% RSLogix 500 project JOB 13 UN FIN_BAK035.RSS, saved by version 10.00.00.00 %
PROJECT "ML06B"    % processor: Bul.1763 MicroLogix 1100 Series B %

PROGRAM FILES
  LAD 2   13 rungs

DATA FILES
  O0 OUTPUT  4 elements
  I1 INPUT  6 elements
  S2 STATUS  66 elements
  B3 BINARY  1 elements
  T4 TIMER  1 elements
  C5 COUNTER  1 elements
  R6 CONTROL  1 elements
  N7 INTEGER  1 elements
  F8 FLOAT  1 elements

LADDER 2
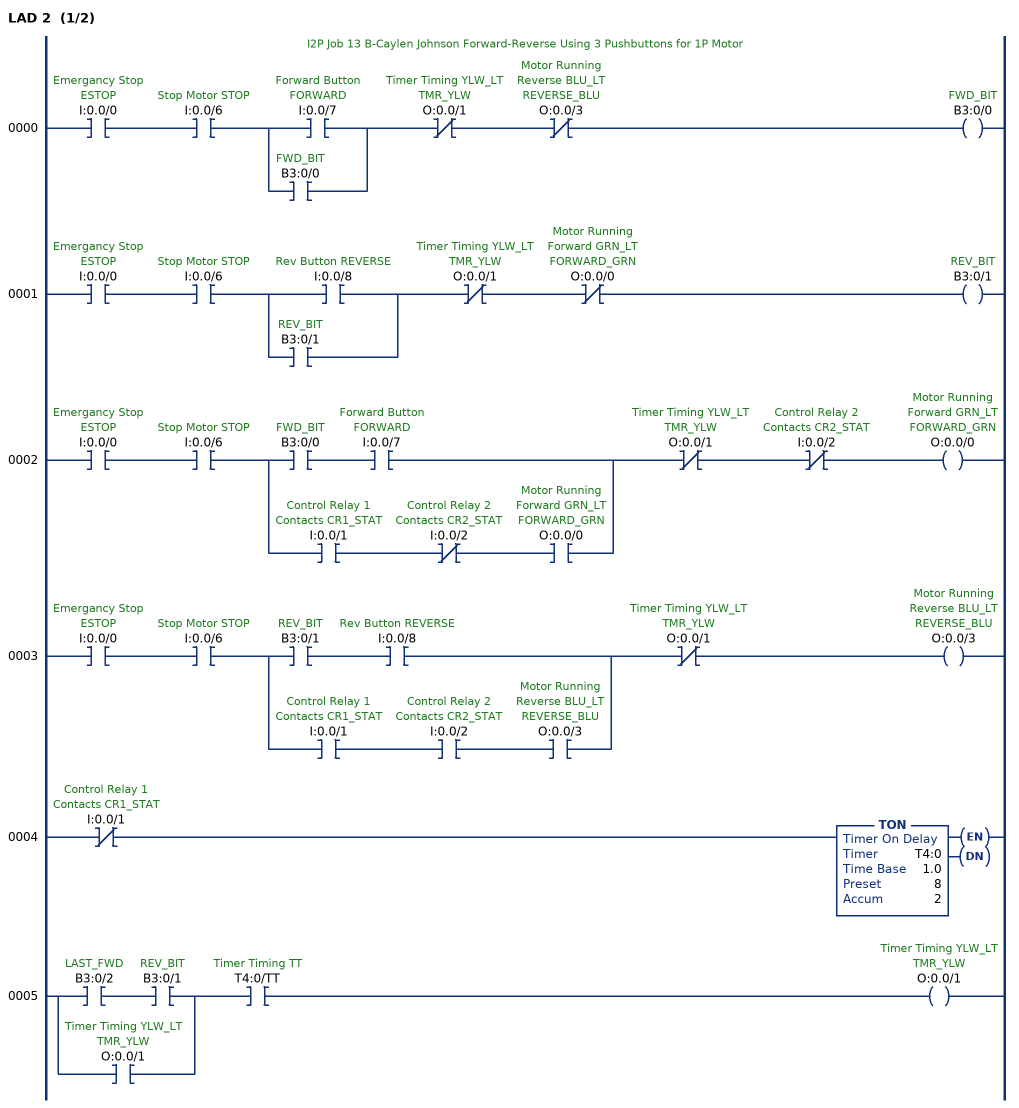
% Rung: 0 %  % edit flag set %
% I2P Job 13 B-Caylen Johnson Forward-Reverse Using 3 Pushbuttons for 1P Motor %
SOR XIC I:0.0/0 XIC I:0.0/6 BST XIC I:0.0/7 NXB XIC B3:0/0 BND XIO O:0.0/1 XIO O:0.0/3 OTE B3:0/0 EOR
%   I:0.0/0  ESTOP  "Emergancy Stop" %
%   I:0.0/6  STOP  "Stop Motor" %
%   I:0.0/7  FORWARD  "Forward Button" %
%   B3:0/0  FWD_BIT %
%   O:0.0/1  TMR_YLW  "Timer Timing YLW_LT" %
%   O:0.0/3  REVERSE_BLU  "Motor Running Reverse BLU_LT" %
% Rung: 1 %
SOR XIC I:0.0/0 XIC I:0.0/6 BST XIC I:0.0/8 NXB XIC B3:0/1 BND XIO O:0.0/1 XIO O:0.0/0 OTE B3:0/1 EOR
%   I:0.0/0  ESTOP  "Emergancy Stop" %
%   I:0.0/6  STOP  "Stop Motor" %
%   I:0.0/8  REVERSE  "Rev Button" %
%   B3:0/1  REV_BIT %
%   O:0.0/1  TMR_YLW  "Timer Timing YLW_LT" %
%   O:0.0/0  FORWARD_GRN  "Motor Running Forward GRN_LT" %
% Rung: 2 %
SOR XIC I:0.0/0 XIC I:0.0/6 BST XIC B3:0/0 XIC I:0.0/7 NXB XIC I:0.0/1 XIO I:0.0/2 XIC O:0.0/0 BND XIO O:0.0/1 XIO I:0.0/2 OTE O:0.0/0 EOR
%   I:0.0/0  ESTOP  "Emergancy Stop" %
%   I:0.0/6  STOP  "Stop Motor" %
%   B3:0/0  FWD_BIT %
%   I:0.0/7  FORWARD  "Forward Button" %
%   I:0.0/1  CR1_STAT  "Control Relay 1 Contacts" %
%   I:0.0/2  CR2_STAT  "Control Relay 2 Contacts" %
%   O:0.0/0  FORWARD_GRN  "Motor Running Forward GRN_LT" %
%   O:0.0/1  TMR_YLW  "Timer Timing YLW_LT" %
% Rung: 3 %
SOR XIC I:0.0/0 XIC I:0.0/6 BST XIC B3:0/1 XIC I:0.0/8 NXB XIC I:0.0/1 XIC I:0.0/2 XIC O:0.0/3 BND XIO O:0.0/1 OTE O:0.0/3 EOR
%   I:0.0/0  ESTOP  "Emergancy Stop" %
%   I:0.0/6  STOP  "Stop Motor" %
%   B3:0/1  REV_BIT %
%   I:0.0/8  REVERSE  "Rev Button" %
%   I:0.0/1  CR1_STAT  "Control Relay 1 Contacts" %
%   I:0.0/2  CR2_STAT  "Control Relay 2 Contacts" %
%   O:0.0/3  REVERSE_BLU  "Motor Running Reverse BLU_LT" %
%   O:0.0/1  TMR_YLW  "Timer Timing YLW_LT" %
% Rung: 4 %
SOR XIO I:0.0/1 TON T4:0 1.0 8 2 EOR
%   I:0.0/1  CR1_STAT  "Control Relay 1 Contacts" %
% Rung: 5 %
SOR BST XIC B3:0/2 XIC B3:0/1 NXB XIC O:0.0/1 BND XIC T4:0/TT OTE O:0.0/1 EOR
%   B3:0/2  LAST_FWD %
%   B3:0/1  REV_BIT %
%   O:0.0/1  TMR_YLW  "Timer Timing YLW_LT" %
%   T4:0/TT  TT  "Timer Timing" %

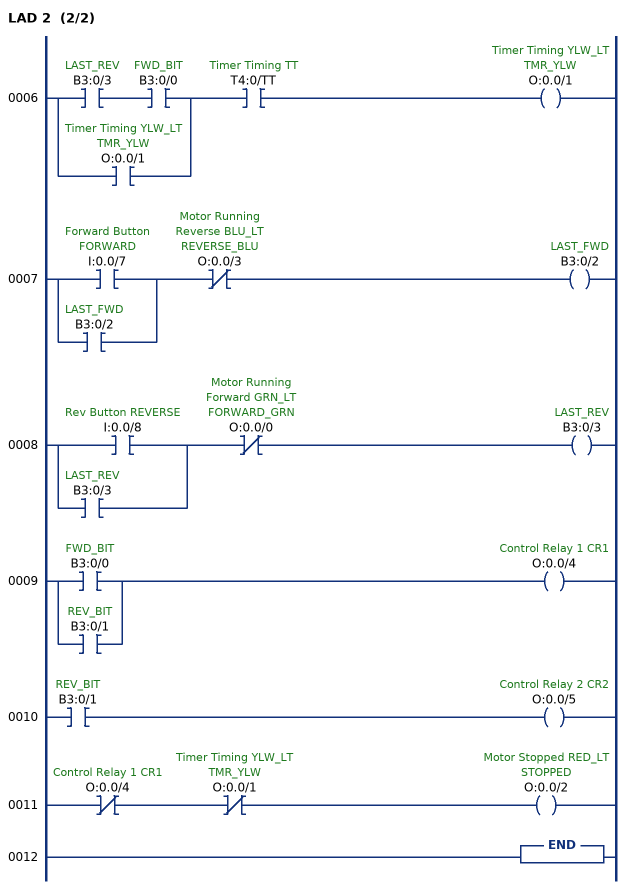
% Rung: 6 %
SOR BST XIC B3:0/3 XIC B3:0/0 NXB XIC O:0.0/1 BND XIC T4:0/TT OTE O:0.0/1 EOR
%   B3:0/3  LAST_REV %
%   B3:0/0  FWD_BIT %
%   O:0.0/1  TMR_YLW  "Timer Timing YLW_LT" %
%   T4:0/TT  TT  "Timer Timing" %
% Rung: 7 %
SOR BST XIC I:0.0/7 NXB XIC B3:0/2 BND XIO O:0.0/3 OTE B3:0/2 EOR
%   I:0.0/7  FORWARD  "Forward Button" %
%   B3:0/2  LAST_FWD %
%   O:0.0/3  REVERSE_BLU  "Motor Running Reverse BLU_LT" %
% Rung: 8 %
SOR BST XIC I:0.0/8 NXB XIC B3:0/3 BND XIO O:0.0/0 OTE B3:0/3 EOR
%   I:0.0/8  REVERSE  "Rev Button" %
%   B3:0/3  LAST_REV %
%   O:0.0/0  FORWARD_GRN  "Motor Running Forward GRN_LT" %
% Rung: 9 %
SOR BST XIC B3:0/0 NXB XIC B3:0/1 BND OTE O:0.0/4 EOR
%   B3:0/0  FWD_BIT %
%   B3:0/1  REV_BIT %
%   O:0.0/4  CR1  "Control Relay 1" %
% Rung: 10 %
SOR XIC B3:0/1 OTE O:0.0/5 EOR
%   B3:0/1  REV_BIT %
%   O:0.0/5  CR2  "Control Relay 2" %
% Rung: 11 %
SOR XIO O:0.0/4 XIO O:0.0/1 OTE O:0.0/2 EOR
%   O:0.0/4  CR1  "Control Relay 1" %
%   O:0.0/1  TMR_YLW  "Timer Timing YLW_LT" %
%   O:0.0/2  STOPPED  "Motor Stopped RED_LT" %
% Rung: 12 %
SOR END EOR

OTHER DOCUMENTED ADDRESSES
  I:0.0/3  3PSS_FWD  "Three Position Selector Switch Forward Direction"
  I:0.0/4  3PSS_REV  "Three Position Selector Switch Reverse Position"
  I:0.0/5  2PSS_A  "Two Position Selector Switch A Position"

DATA TABLE (non-zero values as saved)
DATA B3
% B3:0 % 0X0008
DATA T4
% .PRE .ACC %
% T4:0 % 8 2
